FUNCTION_BLOCK TcoTask_DownCounter EXTENDS TcoCore.TcoTask
VAR
    _SetUpValue : LINT;
    _CounterValue : LINT := -1;
    _InvokeCounter : LINT;
    _DoneCounter : LINT;
END_VAR

IF (THIS^._taskState = eTaskState.Requested) THEN
    CounterValue := SetUpValue;
    _InvokeCounter := _InvokeCounter + 1;
END_IF;

IF (Execute()) THEN
    _CounterValue := _CounterValue - 1;
    DoneWhen(_CounterValue <= 0);
END_IF

IF (THIS^._taskState = eTaskState.Done) THEN
    _DoneCounter := _DoneCounter + 1;
END_IF;

PROPERTY CounterValue : LINT
GET
CounterValue := _CounterValue;
END_GET
SET
_CounterValue := CounterValue;
END_SET
END_PROPERTY

PROPERTY InTheMiddle : BOOL
GET
InTheMiddle := ABS(_SetUpValue - 2 * _CounterValue) < 1;
END_GET
END_PROPERTY

PROPERTY SetUpValue : LINT
GET
SetUpValue := _SetUpValue;
END_GET
SET
_SetUpValue := SetUpValue;
END_SET
END_PROPERTY

END_FUNCTION_BLOCK

(* stored: Version 1.1.0.1
   POU TcoTask_DownCounter: Id {c9c30b05-eaa1-0ec0-3647-f4b645f55955}, SpecialFunc None
   Property CounterValue: Id {5e44ac19-9866-08dc-06d6-6414f4d6a2d7}
   Get Get: Id {0c279010-926b-062b-20f2-4210737e768e}
   Set Set: Id {6b19ab02-0935-003e-244d-bbb8c71f269f}
   Property InTheMiddle: Id {9867b082-7002-0aa1-3a4d-c715e5d40d64}
   Get Get: Id {acd5cc86-cedb-02d0-01d7-1c5c87aa3ae3}
   Property SetUpValue: Id {c15707f7-7428-0efb-3bc4-bb7b3d64a0ed}
   Get Get: Id {845c5d53-9965-06ae-3a07-28f59a824314}
   Set Set: Id {9a3d6377-2d6a-06b3-2191-f8adaf5df528} *)
